FUNCTION_BLOCK fb_WriteData
VAR_INPUT
	bExecute		: BOOL;
	sFileName		: Tc2_System.T_MaxString; (* filename and ending *)
	psData			: POINTER TO STRING(32767);
END_VAR
VAR_OUTPUT
	bBusy				: BOOL;
	bDone				: BOOL;
	bError			: BOOL;
END_VAR
VAR
	diStep			: DINT;
	udiCounter	: UDINT;

	fbFileOpen		: Tc2_System.FB_FileOpen;
	fbFileWrite		: Tc2_System.FB_FileWrite;
	fbFileClose		: Tc2_System.FB_FileClose;

	sTimeStart		: STRING;
	sTimeEnd			: STRING;
END_VAR

udiCounter := udiCounter + 1;

(* pointer check *)
IF (psData = 0)
THEN
	RETURN;
END_IF

IF NOT bExecute
THEN
	diStep := 0;
END_IF

CASE diStep OF

	0:
		fbFileOpen.bExecute		:= FALSE;
		fbFileWrite.bExecute	:= FALSE;
		fbFileClose.bExecute	:= FALSE;
		bBusy := FALSE;
		bDone := FALSE;
		IF bExecute
		THEN
			sTimeStart := GVL_AXIS_CTRL.gfbLocalTime.sLocalTime;
			bBusy  := TRUE;
			diStep := 10;
		END_IF

	10:
		fbFileOpen.bExecute  := TRUE;
		IF fbFileOpen.bBusy
		THEN
			diStep := 20;
		END_IF

	20:
		IF NOT fbFileOpen.bBusy
		THEN
			fbFileOpen.bExecute  := FALSE;
			fbFileWrite.bExecute := TRUE;
			diStep := 30;
		END_IF

	30:
		IF fbFileWrite.bBusy
		THEN
			diStep := 40;
		END_IF

	40:
		IF NOT fbFileWrite.bBusy
		THEN
			fbFileWrite.bExecute := FALSE;
			fbFileClose.bExecute := TRUE;
			diStep := 50;
		END_IF

	50:
		IF fbFileClose.bBusy
		THEN
			diStep := 60;
		END_IF

	60:
		IF NOT fbFileClose.bBusy
		THEN
			fbFileClose.bExecute := FALSE;
			sTimeEnd 	:= GVL_AXIS_CTRL.gfbLocalTime.sLocalTime;
			diStep 		:= 100;
		END_IF
	
	100:
		bBusy := FALSE;
		bDone := TRUE;
END_CASE


fbFileOpen(
	sNetId:= , 
	sPathName:= sFileName, 
	nMode:= FOPEN_MODEAPPEND, 
	ePath:= PATH_GENERIC, 
	bExecute:= , 
	tTimeout:= T#10S, 
	bBusy=> , 
	bError=> , 
	nErrId=> , 
	hFile=> );

fbFileWrite(
	sNetId:= , 
	hFile:= fbFileOpen.hFile, 
	pWriteBuff:= psData, 
	cbWriteLen:= f_Len(psData), 
	bExecute:= , 
	tTimeout:= T#10S, 
	bBusy=> , 
	bError=> , 
	nErrId=> , 
	cbWrite=> );

fbFileClose(
	sNetId:= , 
	hFile:= fbFileOpen.hFile, 
	bExecute:= , 
	tTimeout:= T#10S, 
	bBusy=> , 
	bError=> , 
	nErrId=> );

bError := fbFileOpen.bError OR fbFileWrite.bError;

END_FUNCTION_BLOCK

(* stored: Version 1.1.0.1, ProductVersion 3.1.4024.4
   POU fb_WriteData: Id {f3f927f4-3f6b-4182-9553-c719b7c1ed59}, SpecialFunc None *)
